(* CODESYS project CtaSysEvent_1.0.0.0.library
   Description: Event Library der CTA
   Version: 1.0.0.0
   Title: CtaSysEvent
   Author: SIS
   LanguageModelAttribute: qualified-access-only
   DocFormat: reStructuredText
   Placeholder: CtaSysEvent
   DefaultNamespace: CtaSysEvent
   CompiledLibraryCompatibilityVersion: CODESYS V3.5 SP16 Patch 3
   Company: CTA

Project tree, tasks and I/O mapping:
  libraries: CmpEventMgr, 3.5.17.0 (System); SysTypes2 Interfaces, * (System); Standard, 3.5.18.0 (System); CmpApp, 3.5.17.0 (System); StringUtils, 3.5.18.0 (System); VisuSymbols, 4.5.0.0 (System)
  40 Visualizations/
  30 Program Organization Units/
    function block fbAppEvent [ST]: EventCallback, FB_Init, FB_Exit
    function fcRegistry [ST]
  00000000-0000-0000-0000-000000000000|D:\CoDeSys\LibrariesV3\trunk\Intern\CAA\CAA Template\3.4.0.0 draft\Placeholder.xml
  00000000-0000-0000-0000-000000000000|D:\CoDeSys\LibrariesV3\trunk\Intern\CAA\CAA Template\3.2.0.3 draft\Prefix.pdf
  00000000-0000-0000-0000-000000000000|D:\CoDeSys\LibrariesV3\trunk\Intern\CAA\CAA Template\3.5.2.0 draft\Placeholder.xml
  20 Structs/
  50 Images/
  10 Documenation/
    global variables VersionHistory
    global variables readMe
  21 Interface/
    interface ITF_APPEVENT: proIsRegistred, metStartDone, metPrepeareStop, proDenyStop, metCyclicCall
  11 Library Parameter/
    global variables Parameter
  12 Konstanten/
  60 Textlisten/
  13 Globale Variablen/
    global variables GVL_AppEvent
*)

// 10 Documenation/VersionHistory
(* 

.. image:: ../../Images/CTA_Logo.jpg
   :align: right
   :width: 15% 

**Vorlage**   


============ =========== =========== ============================================
**Date**     **Version** **Author**  **Change**
------------ ----------- ----------- --------------------------------------------
04.03.2021   0.0.0.0     SIS         Vorlage erstellt

============ =========== =========== ============================================


*)
VAR_GLOBAL
    stInfo : STRING:= '0.0.0.0, Vorlage, CTA';
END_VAR

// 10 Documenation/readMe
(*

**ReadMe**
 
|	**Empfehlung**
|
|	Dokumentrieren Sie die Library für eine nachhaltige Entwicklung
|     
| *Beispiel*
| 
| Dies ist die Vorlage Library der CTA. Erstellen Sie ihre Library anhand dieser Vorlage.
*)

VAR_GLOBAL
    xReadMeDone              :   BOOL;
END_VAR

// 13 Globale Variablen/GVL_AppEvent
// {attribute 'hide'}
{attribute 'qualified_only'}
{attribute 'linkalways'}
VAR_GLOBAL
    fbAppEvent          :   fbAppEvent;
    {attribute 'hide'}
    {attribute 'no_init'}
    ayEventInterface    : ARRAY[0..Parameter.uiMaxArray] OF ITF_APPEVENT;
    {attribute 'hide'}
    {attribute 'no_init'}
    diRegistryPlace     : DINT;
END_VAR

// 11 Library Parameter/Parameter
{attribute 'qualified_only'}
VAR_GLOBAL CONSTANT
    uiMaxArray      : UINT := 1000;
END_VAR

// 21 Interface/ITF_APPEVENT
INTERFACE ITF_APPEVENT EXTENDS __SYSTEM.IQueryInterface

PROPERTY proIsRegistred : BOOL
SET
END_SET
GET
END_GET
END_PROPERTY

METHOD metStartDone : BOOL
VAR_INPUT
END_VAR
END_METHOD

METHOD metPrepeareStop : BOOL
VAR_INPUT
END_VAR
END_METHOD

PROPERTY proDenyStop : BOOL
GET
END_GET
END_PROPERTY

METHOD metCyclicCall : BOOL
VAR_INPUT
END_VAR
END_METHOD

END_INTERFACE

// 30 Program Organization Units/fbAppEvent
{attribute 'hide'}
FUNCTION_BLOCK fbAppEvent IMPLEMENTS CmpEventMgr.ICmpEventCallback
VAR_OUTPUT
   udiStartDone     : UDINT;
   udiStopDone      : UDINT;
   udiLogin         : UDINT;
END_VAR
VAR
   hEventStart          : SysTypes.RTS_IEC_HANDLE;
   hInterfaceStart      : SysTypes.RTS_IEC_HANDLE;
   hEventStop           : SysTypes.RTS_IEC_HANDLE;   
   hInterfaceStop       : SysTypes.RTS_IEC_HANDLE;
   hEventCycle          : SysTypes.RTS_IEC_HANDLE; 
   hInterfaceCycle      : SysTypes.RTS_IEC_HANDLE;   
   hEventDenyStop       : SysTypes.RTS_IEC_HANDLE;    
   hInterfaceDenyStop   : SysTypes.RTS_IEC_HANDLE;    
   iecResult            : SysTypes.RTS_IEC_RESULT;
   itfEvtCallback       : CmpEventMgr.ICmpEventCallback;
   pCyclePAram          : POINTER TO EVTPARAM_CmpAppDenyStop;
   _dwStopReason        : DWORD;
  _sAppName             : STRING;
   APP                  : POINTER TO APPLICATION;
   xTryToStop           : BOOL;
   xTryReset            : BOOL;
   xStartDone           : BOOL;
   diDenyStop           : DINT;   
   diEventType          : DINT;
   TON_Cycle            : TON;
   tCycleTime           : TIME;
   tCodeTime            : TIME;
END_VAR

{attribute 'm4export_hide'}
(* The interface ICmpEventCallback must be registered for an event. If this event is posted, this callback method is called.*)
METHOD EventCallback : SysTypes.RTS_IEC_RESULT
VAR_INPUT
	(*Pointer to the event parameters, see Struct EventParam*)
	pEventParam	: POINTER TO EventParam;
END_VAR
VAR
    pStartParam : POINTER TO EVTPARAM_CmpApp;
    pStopParam  : POINTER TO EVTPARAM_CmpAppStop;
    pLoginParam : POINTER TO EVTPARAM_CmpAppComm;

    diFor       : DINT;
    RESULT      : RTS_IEC_RESULT;
END_VAR
APP := AppGetCurrent(ADR(RESULT));
(* Event Handling*)
CASE pEventParam^.EventId OF
    (* Event Start*)
    CmpApp.EventIDs.EVT_StartDone:
        FOR diFor := 0 TO GVL_AppEvent.diRegistryPlace-1 DO
            IF GVL_AppEvent.ayEventInterface[diFor] <> 0 THEN
                GVL_AppEvent.ayEventInterface[diFor].metStartDone();
			END_IF;
		END_FOR;
        pStartParam := pEventParam^.pParameter;
        IF pStartParam <> 0 THEN
            StrCpyA(ADR(_sAppName), SIZEOF(_sAppName), ADR(pStartParam^.pApp^.szName));
        END_IF
        udiStartDone := udiStartDone + 1;
        xStartDone   := TRUE;
    (* Event DenyStop *)
    CmpApp.EventIDs.EVT_DenyStop:
        pCyclePAram := pEventParam^.pParameter;
        diEventType := EventGetEvent(pCyclePAram^.ulStopReason);
        diDenyStop := 0;
        FOR diFor := 0 TO GVL_AppEvent.diRegistryPlace -1 DO
            IF GVL_AppEvent.ayEventInterface[diFor] <> 0 THEN
                IF GVL_AppEvent.ayEventInterface[diFor].proDenyStop THEN
                    diDenyStop := diDenyStop + 1;        
				END_IF;
			END_IF;
		END_FOR;
        IF diDenyStop > 0 AND diEventType <> CmpApp.EventIDs.EVTVERSION_CmpAppException THEN
            pCyclePAram^.bDeny := 1;
            IF diEventType = CmpApp.EventIDs.EVTVERSION_CmpAppReset THEN
                xTryReset  := TRUE;    
            ELSE
                xTryToStop := TRUE;    
			END_IF   
        ELSE
            pCyclePAram^.bDeny  := 0;
            xTryToStop          := TRUE; 
            diDenyStop          := 0;
        END_IF;               
    (* COM Cycle *)
    CmpApp.EventIDs.EVT_CommCycle:
        TON_Cycle();
        tCycleTime := TON_Cycle.ET;
        TON_Cycle.IN := FALSE;       
        TON_Cycle();
        TON_Cycle.IN := TRUE;
        TON_Cycle.PT := T#30S;
        TON_Cycle();
        diDenyStop := 0;
        FOR diFor := 0 TO GVL_AppEvent.diRegistryPlace -1 DO
            IF GVL_AppEvent.ayEventInterface[diFor] <> 0 THEN
                GVL_AppEvent.ayEventInterface[diFor].metCyclicCall();
                IF GVL_AppEvent.ayEventInterface[diFor].proDenyStop THEN
                    diDenyStop := diDenyStop + 1;        
				END_IF;
			END_IF;
		END_FOR;
        IF xTryReset AND diDenyStop = 0 THEN
            CmpApp.AppReset(APP,0);
            xTryReset := FALSE;
            xTryToStop := FALSE;
        END_IF;          
        IF xTryToStop AND diDenyStop = 0 THEN
            CmpApp.AppStopApplication(APP);
            xTryToStop := FALSE;
        END_IF;      
        TON_Cycle(); 
        tCodeTime := TON_Cycle.ET;      
    (* Event Stop*)    
    CmpApp.EventIDs.EVT_PrepareStop: 
        FOR diFor := 0 TO GVL_AppEvent.diRegistryPlace-1 DO
            IF GVL_AppEvent.ayEventInterface[diFor] <> 0 THEN
                GVL_AppEvent.ayEventInterface[diFor].metPrepeareStop();
            END_IF;
        END_FOR;
        pStopParam := pEventParam^.pParameter;    
        IF pStopParam <> 0 THEN
            _dwStopReason := pStopParam^.ulStopReason;
        END_IF
        udiStopDone := udiStopDone + 1;      
END_CASE
END_METHOD

//FB_Init ist immer implizit verfügbar und wird primär für die Initialisierung verwendet.
//Der Rückgabewert wird nicht ausgewertet. Für gezielte Einflussnahme können Sie
//die Methoden explizit deklarieren und darin mit dem Standard-Initialisierungscode 
//zusätzlichen Code bereitstellen. Sie können den Rückgabewert auswerten.
METHOD FB_Init: BOOL
VAR_INPUT    
bInitRetains: BOOL; // TRUE: Die Retain-Variablen werden initialisiert (Reset warm / Reset kalt)    
bInCopyCode: BOOL;  // TRUE: Die Instanz wird danach in den Kopiercode kopiert (Online-Change)
END_VAR
(* Events Registrieren *)
itfEvtCallback      := THIS^;
hEventStart         := EventOpen(CmpApp.EventIds.EVT_StartDone, CmpApp.EventIds.CMPID_CmpApp, iecResult);
hEventStop          := EventOpen(CmpApp.EventIds.EVT_PrepareStop, CmpApp.EventIds.CMPID_CmpApp, iecResult);
hEventCycle         := EventOpen(CmpApp.EventIds.EVT_CommCycle , CmpApp.EventIds.CMPID_CmpApp, iecResult);
hEventDenyStop      := EventOpen(CmpApp.EventIds.EVT_DenyStop , CmpApp.EventIds.CMPID_CmpApp, iecResult);

hInterfaceStart     := EventRegisterCallback(hEventStart, itfEvtCallback, iecResult); 
hInterfaceStop      := EventRegisterCallback(hEventStop, itfEvtCallback, iecResult);
hInterfaceCycle     := EventRegisterCallback(hEventCycle, itfEvtCallback, iecResult);
hInterfaceDenyStop  := EventRegisterCallback(hEventDenyStop, itfEvtCallback, iecResult);
END_METHOD

//FB_Exit muss explizit implementiert werden. Wenn es eine Implementierung gibt, dann wird 
//die Methode aufgerufen, bevor die Steuerung den Code der Funktionsbaustein-Instanz entfernt
//(impliziter Aufruf. Der Rückgabewert wird nicht ausgewertet.
METHOD FB_Exit: BOOL
VAR_INPUT    
bInCopyCode: BOOL;  // TRUE: Die Exit-Methode wird aufgerufen, um die Instanz zu verlassen, die hinterher kopiert wird Online-Change).  
END_VAR
(* Events Löschen *)
EventUnregisterCallback(hEventStart, hInterfaceStart);
EventUnregisterCallback(hEventStop, hInterfaceStop);
EventUnregisterCallback(hEventCycle, hInterfaceCycle);
EventUnregisterCallback(hEventDenyStop, hInterfaceDenyStop);
EventClose2(hEventStart);
EventClose2(hEventStop);
EventClose2(hEventCycle);
EventClose2(hEventDenyStop);
GVL_AppEvent.diRegistryPlace := 0;
END_METHOD

END_FUNCTION_BLOCK

// 30 Program Organization Units/fcRegistry
FUNCTION fcRegistry 
VAR_INPUT
    itfApplicationEventIn   :   ITF_APPEVENT;
END_VAR
VAR
    diCurrentRegitry    :   DINT;
END_VAR

IF itfApplicationEventIn <> 0 THEN 
    diCurrentRegitry := __XADD(ADR(GVL_AppEvent.diRegistryPlace),1);
    IF diCurrentRegitry <= Parameter.uiMaxArray THEN
        IF NOT itfApplicationEventIn.proIsRegistred THEN
            GVL_AppEvent.ayEventInterface[diCurrentRegitry] := itfApplicationEventIn;
            GVL_AppEvent.ayEventInterface[diCurrentRegitry].proIsRegistred := TRUE;
        ELSE
            diCurrentRegitry := __XADD(ADR(GVL_AppEvent.diRegistryPlace),-1);    
        END_IF;   
    END_IF;
END_IF;

END_FUNCTION
